TEXTLIST CoorSys
  1 = 'robot'
  2 = 'couch'
  3 = 'calibration'
  4 = 'spare'
  5 = 'default'
   = ''
END_TEXTLIST

(* stored: Version 1.1.0.1, ProductVersion 3.1.4024.10
   TextList CoorSys: Id {dcc008cd-2da0-4935-878a-e69e7a5aadbc} *)
